ABB RAPID module: Module1.mod

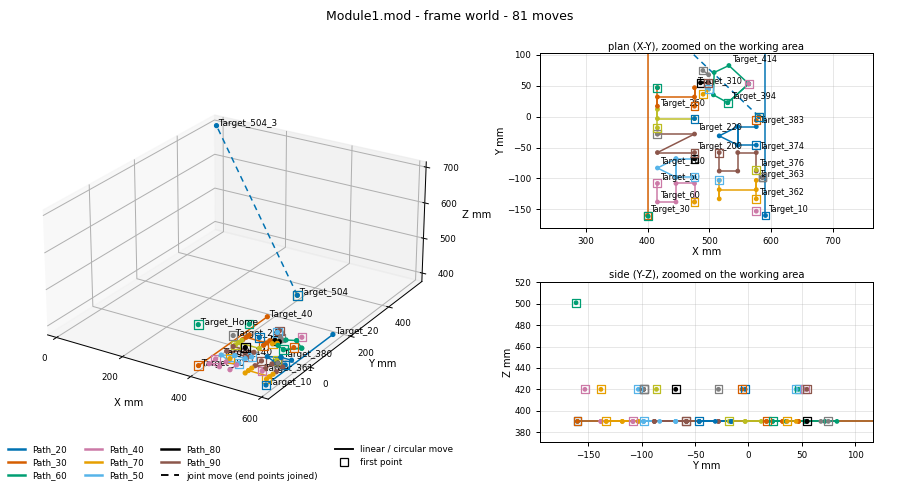
[picture p0: tool path of Module1.mod in frame world, 81 of 81 moves have a stored position in this frame; points joined in program order, loops and branches not executed]
MODULE Module1
    CONST robtarget Target_Home:=[[1.197811499,-1.365906838,111.038482082],[0,0,1,0],[0,0,0,0],[9E+09,9E+09,9E+09,9E+09,9E+09,9E+09]];

    CONST robtarget Target_10:=[[191,0,0],[0,0,1,0],[0,0,0,0],[9E+09,9E+09,9E+09,9E+09,9E+09,9E+09]];
    CONST robtarget Target_20:=[[191,320,0],[0,0,1,0],[0,0,0,0],[9E+09,9E+09,9E+09,9E+09,9E+09,9E+09]];
    CONST robtarget Target_30:=[[0,0,0],[0,0,1,0],[0,0,0,0],[9E+09,9E+09,9E+09,9E+09,9E+09,9E+09]];
    CONST robtarget Target_40:=[[0,320,0],[0,0,1,0],[0,0,0,0],[9E+09,9E+09,9E+09,9E+09,9E+09,9E+09]];

    CONST robtarget Target_50:=[[16.097,51.917,0],[0,0,1,0],[0,0,0,0],[9E+09,9E+09,9E+09,9E+09,9E+09,9E+09]];
    CONST robtarget Target_60:=[[16.097,21.917,0],[0,0,1,0],[0,0,0,0],[9E+09,9E+09,9E+09,9E+09,9E+09,9E+09]];
    CONST robtarget Target_70:=[[46.097,21.917,0],[0,0,1,0],[0,0,0,0],[9E+09,9E+09,9E+09,9E+09,9E+09,9E+09]];
    CONST robtarget Target_80:=[[46.097,51.917,0],[0,0,1,0],[0,0,0,0],[9E+09,9E+09,9E+09,9E+09,9E+09,9E+09]];
    CONST robtarget Target_90:=[[76.097,51.917,0],[0,0,1,0],[0,0,0,0],[9E+09,9E+09,9E+09,9E+09,9E+09,9E+09]];
    CONST robtarget Target_100:=[[76.097,21.917,0],[0,0,1,0],[0,0,0,0],[9E+09,9E+09,9E+09,9E+09,9E+09,9E+09]];
    CONST robtarget Target_120:=[[76.097,61.917,0],[0,0,1,0],[0,0,0,0],[9E+09,9E+09,9E+09,9E+09,9E+09,9E+09]];
    CONST robtarget Target_130:=[[46.097,61.917,0],[0,0,1,0],[0,0,0,0],[9E+09,9E+09,9E+09,9E+09,9E+09,9E+09]];
    CONST robtarget Target_140:=[[16.097,76.917,0],[0,0,1,0],[0,0,0,0],[9E+09,9E+09,9E+09,9E+09,9E+09,9E+09]];
    CONST robtarget Target_150:=[[46.097,91.917,0],[0,0,1,0],[0,0,0,0],[9E+09,9E+09,9E+09,9E+09,9E+09,9E+09]];
    CONST robtarget Target_160:=[[46.097,61.917,0],[0,0,1,0],[0,0,0,0],[9E+09,9E+09,9E+09,9E+09,9E+09,9E+09]];
    CONST robtarget Target_160_2:=[[76.097,91.917,0],[0,0,1,0],[0,0,0,0],[9E+09,9E+09,9E+09,9E+09,9E+09,9E+09]];
    CONST robtarget Target_170:=[[46.097,91.917,0],[0,0,1,0],[0,0,0,0],[9E+09,9E+09,9E+09,9E+09,9E+09,9E+09]];
    CONST robtarget Target_180:=[[76.097,91.917,0],[0,0,1,0],[0,0,0,0],[9E+09,9E+09,9E+09,9E+09,9E+09,9E+09]];
    CONST robtarget Target_110:=[[76.097,21.917,30],[0,0,1,0],[0,0,0,0],[9E+09,9E+09,9E+09,9E+09,9E+09,9E+09]];
    CONST robtarget Target_190:=[[76.097,91.917,30],[0,0,1,0],[0,0,0,0],[9E+09,9E+09,9E+09,9E+09,9E+09,9E+09]];
    CONST robtarget Target_200:=[[76.097,101.917,0],[0,0,1,0],[0,0,0,0],[9E+09,9E+09,9E+09,9E+09,9E+09,9E+09]];
    CONST robtarget Target_210:=[[16.097,101.917,0],[0,0,1,0],[0,0,0,0],[9E+09,9E+09,9E+09,9E+09,9E+09,9E+09]];
    CONST robtarget Target_220:=[[76.097,131.917,0],[0,0,1,0],[0,0,0,0],[9E+09,9E+09,9E+09,9E+09,9E+09,9E+09]];
    CONST robtarget Target_230:=[[16.097,131.917,0],[0,0,1,0],[0,0,0,0],[9E+09,9E+09,9E+09,9E+09,9E+09,9E+09]];
    CONST robtarget Target_240:=[[16.097,131.917,30],[0,0,1,0],[0,0,0,0],[9E+09,9E+09,9E+09,9E+09,9E+09,9E+09]];
    CONST robtarget Target_250:=[[16.097,141.917,0],[0,0,1,0],[0,0,0,0],[9E+09,9E+09,9E+09,9E+09,9E+09,9E+09]];
    CONST robtarget Target_260:=[[16.097,171.917,0],[0,0,1,0],[0,0,0,0],[9E+09,9E+09,9E+09,9E+09,9E+09,9E+09]];
    CONST robtarget Target_270:=[[16.097,156.917,0],[0,0,1,0],[0,0,0,0],[9E+09,9E+09,9E+09,9E+09,9E+09,9E+09]];
    CONST robtarget Target_280:=[[76.097,156.917,0],[0,0,1,0],[0,0,0,0],[9E+09,9E+09,9E+09,9E+09,9E+09,9E+09]];
    CONST robtarget Target_290:=[[76.097,156.917,30],[0,0,1,0],[0,0,0,0],[9E+09,9E+09,9E+09,9E+09,9E+09,9E+09]];
    CONST robtarget Target_300:=[[76.097,176.917,0],[0,0,1,0],[0,0,0,0],[9E+09,9E+09,9E+09,9E+09,9E+09,9E+09]];
    CONST robtarget Target_310:=[[76.097,206.917,0],[0,0,1,0],[0,0,0,0],[9E+09,9E+09,9E+09,9E+09,9E+09,9E+09]];
    CONST robtarget Target_320:=[[76.097,191.917,0],[0,0,1,0],[0,0,0,0],[9E+09,9E+09,9E+09,9E+09,9E+09,9E+09]];
    CONST robtarget Target_330:=[[16.097,191.917,0],[0,0,1,0],[0,0,0,0],[9E+09,9E+09,9E+09,9E+09,9E+09,9E+09]];
    CONST robtarget Target_340:=[[16.097,176.917,0],[0,0,1,0],[0,0,0,0],[9E+09,9E+09,9E+09,9E+09,9E+09,9E+09]];
    CONST robtarget Target_350:=[[16.097,206.917,0],[0,0,1,0],[0,0,0,0],[9E+09,9E+09,9E+09,9E+09,9E+09,9E+09]];
    CONST robtarget Target_360:=[[16.097,206.917,30],[0,0,1,0],[0,0,0,0],[9E+09,9E+09,9E+09,9E+09,9E+09,9E+09]];
    CONST robtarget Target_361:=[[176.097,6.917,30],[0,0,1,0],[0,0,0,0],[9E+09,9E+09,9E+09,9E+09,9E+09,9E+09]];
    CONST robtarget Target_362:=[[176.097,26.917,0],[0,0,1,0],[0,0,0,0],[9E+09,9E+09,9E+09,9E+09,9E+09,9E+09]];
    CONST robtarget Target_363:=[[176.097,56.917,0],[0,0,1,0],[0,0,0,0],[9E+09,9E+09,9E+09,9E+09,9E+09,9E+09]];
    CONST robtarget Target_364:=[[176.097,41.917,0],[0,0,1,0],[0,0,0,0],[9E+09,9E+09,9E+09,9E+09,9E+09,9E+09]];
    CONST robtarget Target_365:=[[116.097,41.917,0],[0,0,1,0],[0,0,0,0],[9E+09,9E+09,9E+09,9E+09,9E+09,9E+09]];
    CONST robtarget Target_366:=[[116.097,26.917,0],[0,0,1,0],[0,0,0,0],[9E+09,9E+09,9E+09,9E+09,9E+09,9E+09]];
    CONST robtarget Target_367:=[[116.097,56.917,0],[0,0,1,0],[0,0,0,0],[9E+09,9E+09,9E+09,9E+09,9E+09,9E+09]];
    CONST robtarget Target_368:=[[116.097,56.917,30],[0,0,1,0],[0,0,0,0],[9E+09,9E+09,9E+09,9E+09,9E+09,9E+09]];
    CONST robtarget Target_370:=[[116.097,101.917,0],[0,0,1,0],[0,0,0,0],[9E+09,9E+09,9E+09,9E+09,9E+09,9E+09]];
    CONST robtarget Target_371:=[[116.097,71.917,0],[0,0,1,0],[0,0,0,0],[9E+09,9E+09,9E+09,9E+09,9E+09,9E+09]];
    CONST robtarget Target_372:=[[146.097,71.917,0],[0,0,1,0],[0,0,0,0],[9E+09,9E+09,9E+09,9E+09,9E+09,9E+09]];
    CONST robtarget Target_373:=[[146.097,101.917,0],[0,0,1,0],[0,0,0,0],[9E+09,9E+09,9E+09,9E+09,9E+09,9E+09]];
    CONST robtarget Target_375:=[[176.097,71.917,0],[0,0,1,0],[0,0,0,0],[9E+09,9E+09,9E+09,9E+09,9E+09,9E+09]];
    CONST robtarget Target_374:=[[176.097,101.917,0],[0,0,1,0],[0,0,0,0],[9E+09,9E+09,9E+09,9E+09,9E+09,9E+09]];
    CONST robtarget Target_369:=[[186.097,61.917,30],[0,0,1,0],[0,0,0,0],[9E+09,9E+09,9E+09,9E+09,9E+09,9E+09]];
    CONST robtarget Target_376:=[[176.097,73.917,30],[0,0,1,0],[0,0,0,0],[9E+09,9E+09,9E+09,9E+09,9E+09,9E+09]];
    CONST robtarget Target_377:=[[176.097,113.917,0],[0,0,1,0],[0,0,0,0],[9E+09,9E+09,9E+09,9E+09,9E+09,9E+09]];
    CONST robtarget Target_378:=[[146.097,113.917,0],[0,0,1,0],[0,0,0,0],[9E+09,9E+09,9E+09,9E+09,9E+09,9E+09]];
    CONST robtarget Target_379:=[[116.097,128.917,0],[0,0,1,0],[0,0,0,0],[9E+09,9E+09,9E+09,9E+09,9E+09,9E+09]];
    CONST robtarget Target_380:=[[146.097,143.917,0],[0,0,1,0],[0,0,0,0],[9E+09,9E+09,9E+09,9E+09,9E+09,9E+09]];
    CONST robtarget Target_381:=[[146.097,113.917,0],[0,0,1,0],[0,0,0,0],[9E+09,9E+09,9E+09,9E+09,9E+09,9E+09]];
    CONST robtarget Target_382:=[[146.097,143.917,0],[0,0,1,0],[0,0,0,0],[9E+09,9E+09,9E+09,9E+09,9E+09,9E+09]];
    CONST robtarget Target_383:=[[176.097,143.917,0],[0,0,1,0],[0,0,0,0],[9E+09,9E+09,9E+09,9E+09,9E+09,9E+09]];
    CONST robtarget Target_384:=[[176.097,153.917,30],[0,0,1,0],[0,0,0,0],[9E+09,9E+09,9E+09,9E+09,9E+09,9E+09]];
    TASK PERS tooldata MarcadorBonitoTCP:=[TRUE,[[67.462,0,121.762],[0.866025404,0,0.5,0]],[1,[0,0,1],[1,0,0,0],0,0,0]];
    TASK PERS wobjdata Wobj_Bonito:=[FALSE,TRUE,"",[[400,-160,390],[1,0,0,0]],[[0,0,0],[1,0,0,0]]];
    TASK PERS tooldata tool_0 := [TRUE,[[0,0,0],[1,0,0,0]],[1,[0,0,1],[1,0,0,0],0,0,0]];
    CONST robtarget Target_394:=[[129.902,182.615,0],[0,0,1,0],[0,0,0,0],[9E+09,9E+09,9E+09,9E+09,9E+09,9E+09]];
    CONST robtarget Target_404:=[[163.86,213.155,0],[0,0,1,0],[0,0,0,0],[9E+09,9E+09,9E+09,9E+09,9E+09,9E+09]];
    CONST robtarget Target_414:=[[131.777,242.791,0],[0,0,1,0],[0,0,0,0],[9E+09,9E+09,9E+09,9E+09,9E+09,9E+09]];
    CONST robtarget Target_424:=[[107.929,231.546,0],[0,0,1,0],[0,0,0,0],[9E+09,9E+09,9E+09,9E+09,9E+09,9E+09]];
    CONST robtarget Target_434:=[[106.71,195.27,0],[0,0,1,0],[0,0,0,0],[9E+09,9E+09,9E+09,9E+09,9E+09,9E+09]];
    CONST robtarget Target_444:=[[89.996,196.254,0],[0,0,1,0],[0,0,0,0],[9E+09,9E+09,9E+09,9E+09,9E+09,9E+09]];
    CONST robtarget Target_454:=[[98.944,204.642,0],[0,0,1,0],[0,0,0,0],[9E+09,9E+09,9E+09,9E+09,9E+09,9E+09]];
    CONST robtarget Target_464:=[[85.808,214.817,0],[0,0,1,0],[0,0,0,0],[9E+09,9E+09,9E+09,9E+09,9E+09,9E+09]];
    CONST robtarget Target_474:=[[98.506,214.827,0],[0,0,1,0],[0,0,0,0],[9E+09,9E+09,9E+09,9E+09,9E+09,9E+09]];
    CONST robtarget Target_484:=[[89.639,234.781,0],[0,0,1,0],[0,0,0,0],[9E+09,9E+09,9E+09,9E+09,9E+09,9E+09]];
    CONST robtarget Target_494:=[[99.013,227.79,0],[0,0,1,0],[0,0,0,0],[9E+09,9E+09,9E+09,9E+09,9E+09,9E+09]];
    CONST robtarget Target_404_2:=[[163.86,213.155,30],[0,0,1,0],[0,0,0,0],[9E+09,9E+09,9E+09,9E+09,9E+09,9E+09]];
    CONST robtarget Target_454_2:=[[98.944,204.642,30],[0,0,1,0],[0,0,0,0],[9E+09,9E+09,9E+09,9E+09,9E+09,9E+09]];
    CONST robtarget Target_474_2:=[[98.506,214.827,30],[0,0,1,0],[0,0,0,0],[9E+09,9E+09,9E+09,9E+09,9E+09,9E+09]];
    CONST robtarget Target_504:=[[180.72,160.063,169.098],[0,0,1,0],[0,0,0,0],[9E+09,9E+09,9E+09,9E+09,9E+09,9E+09]];
    CONST robtarget Target_504_3:=[[-400,710,310],[0.430459334,-0.560985527,0.560985527,0.430459334],[0,0,-1,0],[9E+09,9E+09,9E+09,9E+09,9E+09,9E+09]];

    PROC main()
       WHILE TRUE DO
           IF DI_01 = 1 THEN
               SetDO INICIAL,1;
                WaitTime 2;
                SetDO INICIAL,0;
                SetDO START,1;
                WaitDI SENSOR,1;
                SetDO START,0;
               SET DO_01;
                Path_60;
                Path_40; !Letra S
                Path_70;
                Path_50; !Letra A
                Path_80;
                Path_90; !Letra N
                Path_100;
                Path_110; !Letra T
                Path_120;
                Path_130; !Letra I
                Path_140;
                Path_145;
                Path_150; !Letra I
                Path_160;
                Path_165;
                Path_170; !Letra S
                Path_180;
                Path_190;
                Path_200; !Letra A
                Path_210;
                Path_220; !Diamante
                Path_260;
                Path_230;
                Path_270;
                Path_240;
                Path_280;
                Path_250;
                Path_60; !Home
                RESET DO_01;
                SetDO START,1;
                WaitTime 10;
                SetDO INICIAL,1;
                SetDO START,0;
           ENDIF
           IF DI_02 = 1 THEN
               SET DO_02;
               Path_300; !Cambio Herramienta
               RESET DO_02;
           ENDIF
       ENDWHILE
    ENDPROC

    PROC Path_20()
        MoveL Target_10,v100,z10,MarcadorBonitoTCP\WObj:=Wobj_Bonito;
        MoveL Target_20,v100,z10,MarcadorBonitoTCP\WObj:=Wobj_Bonito;
    ENDPROC
    PROC Path_30()
        MoveL Target_30,v100,z10,MarcadorBonitoTCP\WObj:=Wobj_Bonito;
        MoveL Target_40,v100,z10,MarcadorBonitoTCP\WObj:=Wobj_Bonito;
    ENDPROC

    PROC Path_60()
        MoveL Target_Home,v100,z10,MarcadorBonitoTCP\WObj:=Wobj_Bonito;
    ENDPROC
    PROC Path_40() !Letra S
        MoveL Target_50,v100,z1,MarcadorBonitoTCP\WObj:=Wobj_Bonito;
        MoveL Target_60,v100,z10,MarcadorBonitoTCP\WObj:=Wobj_Bonito;
        MoveL Target_70,v100,z10,MarcadorBonitoTCP\WObj:=Wobj_Bonito;
        MoveL Target_80,v100,z10,MarcadorBonitoTCP\WObj:=Wobj_Bonito;
        MoveL Target_90,v100,z10,MarcadorBonitoTCP\WObj:=Wobj_Bonito;
        MoveL Target_100,v100,z1,MarcadorBonitoTCP\WObj:=Wobj_Bonito;
    ENDPROC
    PROC Path_70()
        MoveL Target_110,v100,z10,MarcadorBonitoTCP\WObj:=Wobj_Bonito;
    ENDPROC
    PROC Path_50() !Letra A
        MoveL Target_120,v100,z10,MarcadorBonitoTCP\WObj:=Wobj_Bonito;
        MoveL Target_130,v100,z1,MarcadorBonitoTCP\WObj:=Wobj_Bonito;
        MoveL Target_140,v100,z10,MarcadorBonitoTCP\WObj:=Wobj_Bonito;
        MoveL Target_150,v100,z1,MarcadorBonitoTCP\WObj:=Wobj_Bonito;
        MoveL Target_160,v100,z1,MarcadorBonitoTCP\WObj:=Wobj_Bonito;
        MoveL Target_170,v100,z1,MarcadorBonitoTCP\WObj:=Wobj_Bonito;
        MoveL Target_180,v100,z10,MarcadorBonitoTCP\WObj:=Wobj_Bonito;
    ENDPROC
    PROC Path_80()
        MoveL Target_190,v100,z10,MarcadorBonitoTCP\WObj:=Wobj_Bonito;
    ENDPROC
    PROC Path_90() !Letra N
        MoveL Target_200,v100,z10,MarcadorBonitoTCP\WObj:=Wobj_Bonito;
        MoveL Target_210,v100,z10,MarcadorBonitoTCP\WObj:=Wobj_Bonito;
        MoveL Target_220,v100,z10,MarcadorBonitoTCP\WObj:=Wobj_Bonito;
        MoveL Target_230,v100,z10,MarcadorBonitoTCP\WObj:=Wobj_Bonito;
    ENDPROC
    PROC Path_100()
        MoveL Target_240,v100,z10,MarcadorBonitoTCP\WObj:=Wobj_Bonito;
    ENDPROC
    PROC Path_110() !Letra T
        MoveL Target_250,v100,z10,MarcadorBonitoTCP\WObj:=Wobj_Bonito;
        MoveL Target_260,v100,z1,MarcadorBonitoTCP\WObj:=Wobj_Bonito;
        MoveL Target_270,v100,z1,MarcadorBonitoTCP\WObj:=Wobj_Bonito;
        MoveL Target_280,v100,z10,MarcadorBonitoTCP\WObj:=Wobj_Bonito;
    ENDPROC
    PROC Path_120()
        MoveL Target_290,v100,z10,MarcadorBonitoTCP\WObj:=Wobj_Bonito;
    ENDPROC
    PROC Path_130() !Letra I
        MoveL Target_300,v100,z10,MarcadorBonitoTCP\WObj:=Wobj_Bonito;
        MoveL Target_310,v100,z10,MarcadorBonitoTCP\WObj:=Wobj_Bonito;
        MoveL Target_320,v100,z1,MarcadorBonitoTCP\WObj:=Wobj_Bonito;
        MoveL Target_330,v100,z1,MarcadorBonitoTCP\WObj:=Wobj_Bonito;
        MoveL Target_340,v100,z10,MarcadorBonitoTCP\WObj:=Wobj_Bonito;
        MoveL Target_350,v100,z10,MarcadorBonitoTCP\WObj:=Wobj_Bonito;
    ENDPROC
    PROC Path_140()
        MoveL Target_360,v100,z10,MarcadorBonitoTCP\WObj:=Wobj_Bonito;
    ENDPROC
    PROC Path_145()
        MoveL Target_361,v100,z10,MarcadorBonitoTCP\WObj:=Wobj_Bonito;
    ENDPROC
    PROC Path_150() !Letra I
        MoveL Target_362,v100,z10,MarcadorBonitoTCP\WObj:=Wobj_Bonito;
        MoveL Target_363,v100,z10,MarcadorBonitoTCP\WObj:=Wobj_Bonito;
        MoveL Target_364,v100,z1,MarcadorBonitoTCP\WObj:=Wobj_Bonito;
        MoveL Target_365,v100,z1,MarcadorBonitoTCP\WObj:=Wobj_Bonito;
        MoveL Target_366,v100,z10,MarcadorBonitoTCP\WObj:=Wobj_Bonito;
        MoveL Target_367,v100,z10,MarcadorBonitoTCP\WObj:=Wobj_Bonito;
    ENDPROC
    PROC Path_160()
        MoveL Target_368,v100,z10,MarcadorBonitoTCP\WObj:=Wobj_Bonito;
    ENDPROC
    PROC Path_165()
        MoveL Target_369,v100,z10,MarcadorBonitoTCP\WObj:=Wobj_Bonito;
    ENDPROC
    PROC Path_170() !Letra S
        MoveL Target_370,v100,z1,MarcadorBonitoTCP\WObj:=Wobj_Bonito;
        MoveL Target_371,v100,z10,MarcadorBonitoTCP\WObj:=Wobj_Bonito;
        MoveL Target_372,v100,z10,MarcadorBonitoTCP\WObj:=Wobj_Bonito;
        MoveL Target_373,v100,z10,MarcadorBonitoTCP\WObj:=Wobj_Bonito;
        MoveL Target_374,v100,z10,MarcadorBonitoTCP\WObj:=Wobj_Bonito;
        MoveL Target_375,v100,z1,MarcadorBonitoTCP\WObj:=Wobj_Bonito;
    ENDPROC
    PROC Path_180()
        MoveL Target_369,v100,z10,MarcadorBonitoTCP\WObj:=Wobj_Bonito;
    ENDPROC
    PROC Path_190()
        MoveL Target_376,v100,z10,MarcadorBonitoTCP\WObj:=Wobj_Bonito;
    ENDPROC
    PROC Path_200() !Letra A
        MoveL Target_377,v100,z10,MarcadorBonitoTCP\WObj:=Wobj_Bonito;
        MoveL Target_378,v100,z1,MarcadorBonitoTCP\WObj:=Wobj_Bonito;
        MoveL Target_379,v100,z10,MarcadorBonitoTCP\WObj:=Wobj_Bonito;
        MoveL Target_380,v100,z1,MarcadorBonitoTCP\WObj:=Wobj_Bonito;
        MoveL Target_381,v100,z1,MarcadorBonitoTCP\WObj:=Wobj_Bonito;
        MoveL Target_382,v100,z1,MarcadorBonitoTCP\WObj:=Wobj_Bonito;
        MoveL Target_383,v100,z10,MarcadorBonitoTCP\WObj:=Wobj_Bonito;
    ENDPROC
    PROC Path_210()
        MoveL Target_384,v100,z10,MarcadorBonitoTCP\WObj:=Wobj_Bonito;
    ENDPROC
    PROC Path_220() !Diamante
        MoveL Target_394,v100,z1,MarcadorBonitoTCP\WObj:=Wobj_Bonito;
        MoveL Target_404,v100,z1,MarcadorBonitoTCP\WObj:=Wobj_Bonito;
        MoveL Target_414,v100,z1,MarcadorBonitoTCP\WObj:=Wobj_Bonito;
        MoveL Target_424,v100,z1,MarcadorBonitoTCP\WObj:=Wobj_Bonito;
        MoveL Target_434,v100,z1,MarcadorBonitoTCP\WObj:=Wobj_Bonito;
        MoveL Target_394,v100,z1,MarcadorBonitoTCP\WObj:=Wobj_Bonito;
        MoveL Target_404,v100,z1,MarcadorBonitoTCP\WObj:=Wobj_Bonito;
    ENDPROC
    PROC Path_260()
        MoveL Target_404_2,v100,z10,MarcadorBonitoTCP\WObj:=Wobj_Bonito;
    ENDPROC
    PROC Path_230() !Linea1
        MoveL Target_444,v100,z10,MarcadorBonitoTCP\WObj:=Wobj_Bonito;
        MoveL Target_454,v100,z10,MarcadorBonitoTCP\WObj:=Wobj_Bonito;
    ENDPROC
     PROC Path_270()
        MoveL Target_454_2,v100,z10,MarcadorBonitoTCP\WObj:=Wobj_Bonito;
    ENDPROC
    PROC Path_240() !Linea2
        MoveL Target_464,v100,z10,MarcadorBonitoTCP\WObj:=Wobj_Bonito;
        MoveL Target_474,v100,z10,MarcadorBonitoTCP\WObj:=Wobj_Bonito;
    ENDPROC
    PROC Path_280()
        MoveL Target_474_2,v100,z10,MarcadorBonitoTCP\WObj:=Wobj_Bonito;
    ENDPROC
    PROC Path_250() !Linea3
        MoveL Target_484,v100,z10,MarcadorBonitoTCP\WObj:=Wobj_Bonito;
        MoveL Target_494,v100,z10,MarcadorBonitoTCP\WObj:=Wobj_Bonito;
    ENDPROC
    PROC Path_290() !Home
        MoveL Target_504,v100,z10,MarcadorBonitoTCP\WObj:=Wobj_Bonito;
    ENDPROC
    PROC Path_300() !Cambio Herramienta
        MoveL Target_504,v100,z10,MarcadorBonitoTCP\WObj:=Wobj_Bonito;
        MoveJ Target_504_3,v100,z10,tool_0\WObj:=Wobj_Bonito;
    ENDPROC
ENDMODULE
